PROGRAM MAIN
VAR
	myXts : XtsFacade;
END_VAR

END_PROGRAM

(* stored: Version 1.1.0.1, ProductVersion 3.1.4024.12
   POU MAIN: Id {0dbc6255-70d0-4e3f-b01e-75c1fd52a931}, SpecialFunc None *)
